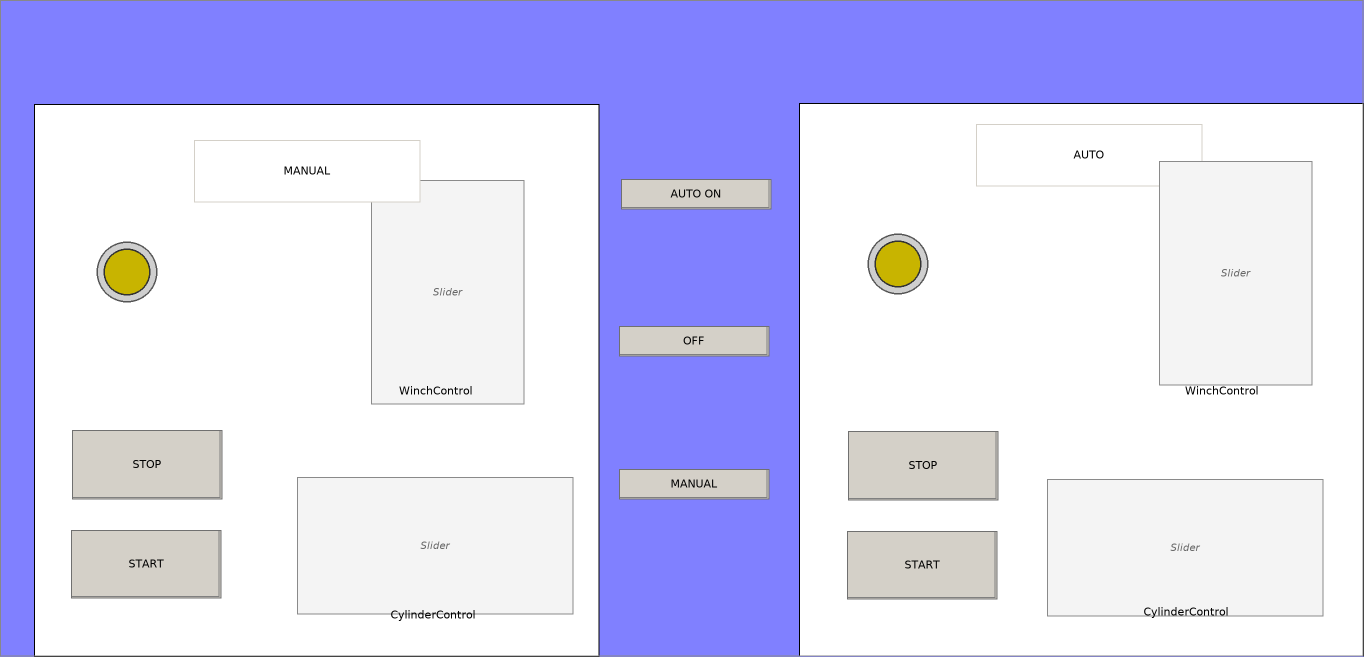
VISUALIZATION HMI_ControlBox  // 1364x657
    Rectangle (34,104 565x553)
    Button (71,530 150x68), "START"
        tap GVL_ControlBox.stControlParams.Start
    Button (72,430 150x69), "STOP"
        tap GVL_ControlBox.stControlParams.Stop
    Slider (297,477 276x137), variable: GVL_ControlBox.stControlParams.JOY_X, scale -1..1
    Slider (371,180 153x224), variable: GVL_ControlBox.stControlParams.JOY_Y, scale -1..1
    Textfield (194,140 226x62), "MANUAL", input disabled if: GVL_ControlBox.stControlParams.Auto
    Rectangle (799,103 565x553)
    Textfield (976,124 226x62), "AUTO", input disabled if: GVL_ControlBox.stControlParams.Manual
    Button (847,531 150x68), "START"
        tap GVL_ControlBox.stControlParams.Start
    Button (848,431 150x69), "STOP"
        tap GVL_ControlBox.stControlParams.Stop
    Slider (1159,161 153x224), variable: GVL_ControlBox.stControlParams.JOY_Y, scale -1..1
    Slider (1047,479 276x137), variable: GVL_ControlBox.stControlParams.JOY_X, scale -1..1
    Lamp1 (92,237 70x70), tooltip "ManualModeOn", variable: GVL_ControlBox.stControlParams.Manual, style: Lamp-Lamp1-Yellow
    Lamp1 (863,229 70x70), tooltip "AutoModeOn", variable: GVL_ControlBox.stControlParams.Auto, style: Lamp-Lamp1-Yellow
    Button (621,179 150x30), "AUTO ON"
    Button (619,326 150x30), "OFF"
    Button (619,469 150x30), "MANUAL"
    Label (1111,597 150x30), "CylinderControl"
    Label (358,600 150x30), "CylinderControl"
    Label (361,376 150x30), "WinchControl"
    Label (1147,376 150x30), "WinchControl"
END_VISUALIZATION

(* stored: Version 1.1.0.1, ProductVersion 3.1.4024.12
   Visu HMI_ControlBox: Id {c601b8de-a6cf-43e9-a9b3-3805307c77d9} *)
